{attribute 'reflection'}
FUNCTION_BLOCK PUBLIC ABSTRACT Fb_ModuleBase
VAR_INPUT
	nModuleID			: 	UDINT 	:= 1 	; // module reference number used for fault, enable, reset, and safety functions (default := 1, 0 = main system)
	// main system Inputs
	bEnable				: 	BOOL	:= FALSE ; // (autolinked) module enable 	
	bCmdReset 			: 	BOOL	:= FALSE ; // (AutoLinked) reset all faults 
	bSysFatalFault		: 	BOOL 	:= FALSE ; // (AutoLinked) System fatal fault active
	bSysCycleFault		: 	BOOL 	:= FALSE ; // (AutoLinked) System fatal fault active 
	bCmdPause			: 	BOOL 	:= FALSE ; // Pause command	bCmdToStart			
	// Internal safety 
	bSafetyOK			: BOOL := FALSE ; // Module internal safety is ok
END_VAR
VAR_OUTPUT
	sName 				: STRING 	:= 'NA' 			; // Module name
	bAddedToSystem		: BOOL 		:= FALSE 			; // module has been added to the system
 	// Com to main system
	fbFaultHandler		: 	Fb_FaultHandler 		; // Fault handler 
	sStateIndicator		: 	STRING := ''			; // Operator message, indication of current step or function 

	// Fault indications
	bMissingCond	: BOOL := FALSE ; // Module missing condition active
	bFatalFault		: BOOL := FALSE ; // Module fatal fault is active
	bCycleFault		: BOOL := FALSE ; // Module cycle fault is active

	// Check values
	bReferenceOk	: BOOL := FALSE ; // All module references  have been checked
	// State indication
	bIsSafe			: BOOL := FALSE ; // Module is safe and locked until safety is ok
	bNoreference	: BOOL := FALSE ; // Module Startup Undefined initialization required
	binitialized	: BOOL := FALSE ; // Module startup initialized waiting for startup command
	bHomed 			: BOOL := FALSE ; // Module startup homed waiting for further further commands

	bHolding 		: BOOL := FALSE ; // Module Module Hold motion command executing
	bHeld	 		: BOOL := FALSE ; // Module Hold Motion is held until command is released	
	
	bResetDone 		: BOOL := FALSE ; // Module reset is done   

	bManual 		: BOOL := FALSE ; // Module Work status Module in Manual
	bSemiAuto		: BOOL := FALSE ; // Module work status in semi automatic
	bStartAuto		: BOOL := FALSE ; // Module start automatic cycle 
	bAutomatic 		: BOOL := FALSE ; // Module Work status Module in Automatic mode
	bPaused			: BOOL := false ; // Module paused
	
	bPoweringOff	: BOOL := FALSE ; // Module is powering off
	bPowerdOff		: BOOL := FALSE ; // Module has powerd off 	

END_VAR
VAR 
	// Internal functions 
	ReCmdReset 			: R_TRIG ;
	// manual functions 
	bParametersAdded	: BOOL := FALSE ;
	// Persistent data
	bCmdWritePersistent : BOOL := FALSE ; // write persistent data to memory
	// Module data
	stMessage			: UDT_Fault			; // Message data
	// Function path 
	{attribute 'instance-path'} 
    {attribute 'noinit'}
	sPath				: STRING	; // Path name of function (used for manual reference)
END_VAR

// Get device name from function
IF sName = 'NA' THEN 
	sName := F_FBNameFromPath(sPath := sPath);
END_IF

// Add module to system
IF NOT bAddedToSystem THEN
	bAddedToSystem S= SystemBase.CmdAddModule(refToModule := THIS^);
	RETURN;
END_IF

IF NOT bReferenceOk THEN 
	bReferenceOk S= CheckReferences();
	RETURN;
ELSE 
	// Execute functions
	ExecMainBaseFunctions();
END_IF

METHOD PROTECTED ABSTRACT CallComponents : BOOL
VAR_INPUT
END_VAR
END_METHOD

METHOD PROTECTED ABSTRACT CheckCollision : BOOL // Checks device commands for positble collisions  and block if necesarry
VAR_INPUT
END_VAR
END_METHOD

METHOD PUBLIC ABSTRACT CheckReferences : BOOL
VAR_INPUT
END_VAR
END_METHOD

METHOD INTERNAL CmdAutomatic : BOOL
VAR_INPUT
END_VAR
IF NOT bAutomatic THEN 
	bStartAuto 		:= TRUE ;
END_IF 

CmdAutomatic 	:= bAutomatic;
END_METHOD

METHOD INTERNAL CmdEstop : BOOL
VAR_INPUT
END_VAR
ExecSafeStop();
bSemiAuto		:= FALSE ;
bAutomatic 		:= FALSE ;

CmdEstop := bIsSafe ;
END_METHOD

METHOD INTERNAL CmdHold : BOOL
VAR_INPUT
END_VAR
ExecHold();


CmdHold := bHeld ;
END_METHOD

METHOD Internal CmdHome : BOOL
VAR_INPUT
END_VAR
ExecHome();

CmdHome := bHomed;
END_METHOD

METHOD INTERNAL CmdInit : BOOL
VAR_INPUT
END_VAR
ExecInit();

CmdInit := binitialized;
END_METHOD

METHOD Internal CmdManual : BOOL
VAR_INPUT
END_VAR
ExecManual();

CmdManual := bManual;
END_METHOD

METHOD INTERNAL CmdPowerOff : BOOL
VAR_INPUT
END_VAR
ExecPowerOff();
bAutomatic := FALSE ;

CmdPowerOff := bPowerdOff;
END_METHOD

METHOD INTERNAL CmdSemiAuto : BOOL
VAR_INPUT
END_VAR
ExecSemiAuto();

CmdSemiAuto := bSemiAuto ;
END_METHOD

METHOD PROTECTED ABSTRACT ExecAutomatic : BOOL
VAR_INPUT
END_VAR
END_METHOD

METHOD PUBLIC ExecBaseFunctions : BOOL
VAR_INPUT
END_VAR
END_METHOD

METHOD ExecFaultHandling : BOOL
VAR_INPUT
END_VAR
// Call message function
	fbFaultHandler(bReset := bCmdReset);

// Call reset functions
	ReCmdReset( CLK := bCmdReset);
	
	IF ReCmdReset.Q THEN 
		bResetDone := FALSE ;
	ELSIF NOT bResetDone THEN 
		fbFaultHandler.bReset := TRUE ;
		bResetDone := ExecReset();
	END_IF
	
	bCmdReset := FALSE ;
// add message if active
	fbFaultHandler.CmdAddFault( stFault := stMessage );

	
	bFatalFault := fbFaultHandler.bActFF ;
	bCycleFault := fbFaultHandler.bActCF ;
	
	IF bFatalFault THEN
		ExecSafeStop()	;
		bHomed			:= FALSE;
	ELSIF bCycleFault THEN
		bHeld			S= ExecHold();
		bHolding 		:= NOT bHeld ;
	END_IF

// Reset safe state when enable is active
	bIsSafe R= bSafetyOK ;

// Prevent automatic start when fault is active
	bStartAuto R= bCmdReset OR bFatalFault OR bCycleFault ;
END_METHOD

METHOD PROTECTED ABSTRACT ExecHold : BOOL
VAR_INPUT
END_VAR
END_METHOD

METHOD PROTECTED ABSTRACT ExecHome : BOOL
VAR_INPUT
END_VAR
END_METHOD

METHOD PROTECTED ABSTRACT ExecInit : BOOL
VAR_INPUT
END_VAR
END_METHOD

METHOD INTERNAL ExecMainBaseFunctions : BOOL
VAR_INPUT
END_VAR
// Call fault handling function 
ExecFaultHandling();

// Check for anny Internal collisions
CheckCollision();

// Call components 
CallComponents();


// Run automatic function 
IF bStartAuto OR bAutomatic THEN 
	bAutomatic 	:= ExecAutomatic();
	bStartAuto 	:= FALSE ;
	bSemiAuto	:= FALSE ;
ELSIF bEnable AND NOT bAutomatic THEN
	bAutomatic 	:= FALSE ;
	bSemIAuto  	:= ExecSemiAuto();
ELSE
	bAutomatic 	:= FALSE ;
	bSemiAuto	:= FALSE ;
END_IF

// run Base Functions 
IF binitialized 
AND bEnable
AND bHomed 
AND NOT bManual THEN 
	ExecBaseFunctions();
END_IF


// Persistent data 
IF bCmdWritePersistent THEN 
	bCmdWritePersistent R= DataManager.FbPersistentManager.Write();
END_IF
END_METHOD

METHOD PROTECTED ExecManual : BOOL
VAR_INPUT
END_VAR
bManual := true;
END_METHOD

METHOD PROTECTED ABSTRACT ExecPowerOff : BOOL
VAR_INPUT
END_VAR
END_METHOD

METHOD PROTECTED ABSTRACT ExecReset : BOOL
VAR_INPUT
END_VAR
END_METHOD

METHOD PROTECTED ABSTRACT ExecSafeStop : BOOL
VAR_INPUT
END_VAR
END_METHOD

METHOD PROTECTED ExecSemiAuto : BOOL
VAR_INPUT
END_VAR
END_METHOD

END_FUNCTION_BLOCK

(* stored: Version 1.1.0.1, ProductVersion 3.1.4024.5
   POU Fb_ModuleBase: Id {e3f07cb2-eb83-4b34-9aad-2d4595c2aa5d}, SpecialFunc None
   Folder Commands: Id {23a18ca6-8b05-47e8-8c4b-aa1afa1e892a}
   Folder Execute: Id {f0dd53fd-6b62-4b4d-9761-2507a7488bb2}
   Folder Private: Id {c399b340-fa14-4baf-a6f6-90d72fec9257}
   Method CallComponents: Id {22be9b1f-00c3-4e1c-90f8-f2ff5645fc88}
   Method CheckCollision: Id {8d738489-b236-4612-b552-096d24330292}
   Method CheckReferences: Id {fd109a63-20a0-4b77-ba3e-d36429660f9a}
   Method CmdAutomatic: Id {12a5af10-cb9c-42e0-8f13-2adc898b5d5a}
   Method CmdEstop: Id {d05300f1-aa34-43f5-a9f7-94f7856dd9ba}
   Method CmdHold: Id {ab17051c-ea15-419f-9ada-82ef46f33e0a}
   Method CmdHome: Id {3a000da5-5c20-4ff2-8583-74c7fae87bc2}
   Method CmdInit: Id {83c2609c-15fb-4eeb-beb4-42411df76941}
   Method CmdManual: Id {7a18f16c-cb69-42f0-ab80-bae80d368991}
   Method CmdPowerOff: Id {c9bd01d3-368e-4423-bb7c-d2899324267d}
   Method CmdSemiAuto: Id {791a75b1-1408-4ba1-a250-3359f3233728}
   Method ExecAutomatic: Id {60275d51-07c9-40b6-9565-a211f029bc96}
   Method ExecBaseFunctions: Id {9ca3b82c-fc59-4a02-b721-3d67056da31e}
   Method ExecFaultHandling: Id {98e653af-0f09-41a0-bb7f-7370a5927e63}
   Method ExecHold: Id {0018095c-5f39-4db3-b3d8-dd0243064ada}
   Method ExecHome: Id {50f16f13-6654-4092-b3f6-5fd77273a5a8}
   Method ExecInit: Id {6bbf633c-be70-4b2b-b0ef-e1874d2714eb}
   Method ExecMainBaseFunctions: Id {e7f3087e-94c4-4f9d-9692-e5a0969e6fe3}
   Method ExecManual: Id {63d94b51-c5c2-4d65-84f7-21d85d57b86f}
   Method ExecPowerOff: Id {ea164508-7b3d-437c-8288-18cdd09bb9f4}
   Method ExecReset: Id {16710407-862f-42d6-b9d2-79f884d2291c}
   Method ExecSafeStop: Id {6444f87d-3200-4afd-ac19-66712355365b}
   Method ExecSemiAuto: Id {6d784c7b-e589-424b-8150-d725f6353df0} *)
